PROGRAM Tests
VAR
END_VAR

Tests_ListAndFactory();
Tests_Udp();

END_PROGRAM

(* stored: Version 1.1.0.1
   POU Tests: Id {5ebf9a52-e6c9-4043-9013-26b310600035}, SpecialFunc None *)
